FUNCTION F_Toggle : BOOL
VAR_IN_OUT
	Flag : BOOL;
END_VAR

Flag     := NOT Flag;
F_Toggle := Flag;

END_FUNCTION

(* stored: Version 1.1.0.1, ProductVersion 3.1.4024.12
   POU F_Toggle: Id {2fd9d643-df72-4f53-bfab-05136b8b1401}, SpecialFunc None *)
